// TIA Portal project "SzablonMASTER_V17" (V17)

(* hardware
DEVICE "S7-1200 station_1"  S7-1200 Station
   slot 0: "Rack_0"  Rack  V1.0
   slot 1: "PLC_1"  CPU 1214C DC/DC/DC  6ES7 214-1AG40-0XB0  V4.1
*)

// ===== PLC "PLC_1"  CPU 1214C DC/DC/DC =====

DATA_BLOCK "IO"   // DB1
{ S7_Optimized_Access := 'TRUE' }
VERSION : 0.1
   VAR
      StartS1 : Bool;
      StopS2 : Bool;
      RESETS3 : Bool;
      CzujnikEtykieciarkaB1 : Bool;
      CzujnikOdrzutB2 : Bool;
      CzujnikZbiornikB3 : Bool;
      CzujnikWieczkaB4 : Bool;
      SystemWizyjnyC1 : Bool;
      WagaC2 : Real;
      EtykieciarkaE1 : Bool;
      ZaworZ1 : Bool;
      SilownikA1 : Bool;
      SilownikA2 : Bool;
      PrzenosnikM1 : Bool;
      KolumnaZielonyH1 : Bool;
      KolumnaZoltyH2 : Bool;
      KolumnaCzerwonyH3 : Bool;
   END_VAR
BEGIN
END_DATA_BLOCK

DATA_BLOCK "ZadanieFinaloweMASTER_DB"   // DB2
{ S7_Optimized_Access := 'TRUE' }
VERSION : 0.1
// stored: InstanceOfName ZadanieFinaloweMASTER
"ZadanieFinaloweMASTER"
BEGIN
   StopS2 := true;
END_DATA_BLOCK

// folder: System blocks/Program resources

DATA_BLOCK "IEC_Timer_0_DB"   // DB3
{ S7_Optimized_Access := 'TRUE' }
AUTHOR : Simatic
FAMILY : IEC
NAME : IEC_TMR
VERSION : 1.0
// stored: InstanceOfName IEC_TIMER
"IEC_TIMER"
BEGIN
END_DATA_BLOCK

DATA_BLOCK "IEC_Timer_1_DB"   // DB4
{ S7_Optimized_Access := 'TRUE' }
AUTHOR : Simatic
FAMILY : IEC
NAME : IEC_TMR
VERSION : 1.0
// stored: InstanceOfName IEC_TIMER
"IEC_TIMER"
BEGIN
END_DATA_BLOCK

DATA_BLOCK "IEC_Timer_0_DB_1"   // DB5
{ S7_Optimized_Access := 'TRUE' }
AUTHOR : Simatic
FAMILY : IEC
NAME : IEC_TMR
VERSION : 1.0
// stored: InstanceOfName IEC_TIMER
"IEC_TIMER"
BEGIN
END_DATA_BLOCK

DATA_BLOCK "IEC_Timer_0_DB_2"   // DB6
{ S7_Optimized_Access := 'TRUE' }
AUTHOR : Simatic
FAMILY : IEC
NAME : IEC_TMR
VERSION : 1.0
// stored: InstanceOfName IEC_TIMER
"IEC_TIMER"
BEGIN
END_DATA_BLOCK

DATA_BLOCK "IEC_Counter_0_DB"   // DB7
{ S7_Optimized_Access := 'TRUE' }
AUTHOR : Simatic
FAMILY : IEC
NAME : CNTR
VERSION : 1.0
// stored: InstanceOfName IEC_COUNTER
"IEC_COUNTER"
BEGIN
END_DATA_BLOCK

DATA_BLOCK "IEC_Timer_0_DB_3"   // DB8
{ S7_Optimized_Access := 'TRUE' }
AUTHOR : Simatic
FAMILY : IEC
NAME : IEC_TMR
VERSION : 1.0
// stored: InstanceOfName IEC_TIMER
"IEC_TIMER"
BEGIN
END_DATA_BLOCK

// folder: (top level)

FUNCTION_BLOCK "ZadanieFinaloweMASTER"   // FB1, LAD
{ S7_Optimized_Access := 'TRUE' }
VERSION : 0.1
   VAR_INPUT
      StartS1 : Bool;
      StopS2 : Bool;
      RESETS3 : Bool;
      CzujnikEtykieciarkaB1 : Bool;
      CzujnikOdrzutB2 : Bool;
      CzujnikZbiornikB3 : Bool;
      CzujnikWieczkaB4 : Bool;
      SystemWizyjnyC1 : Bool;
      WagaC2 : Real;
   END_VAR
   VAR_OUTPUT
      EtykieciarkaE1 : Bool;
      ZaworZ1 : Bool;
      SilownikA1 : Bool;
      SilownikA2 : Bool;
      PrzenosnikM1 : Bool;
      KolumnaZielonyH1 : Bool;
      KolumnaZoltyH2 : Bool;
      KolumnaCzerwonyH3 : Bool;
   END_VAR
   VAR
      Run : Bool;
      Run_edgeP : Bool;
      Run_edgeN : Bool;
      T1_edge : Bool;
      A2_edge : Bool;
      B3_edge : Bool;
      B4_edge : Bool;
      WagaPuls : Bool;
      "WagaPuls edge" : Bool;
      Alarm : Bool;
      DB5_Q_edge : Bool;
   END_VAR
   VAR_TEMP
      T : Real;
      T_high : Real;
      T_Int : Int;
      T_high_Int : Int;
      Alarm_1_5Hz : Bool;
   END_VAR
   VAR_TEMP   // added for the SCL form of the ladder/FBD networks
      _w1 : Bool;
      _w2 : Bool;
   END_VAR
BEGIN

REGION Network 1
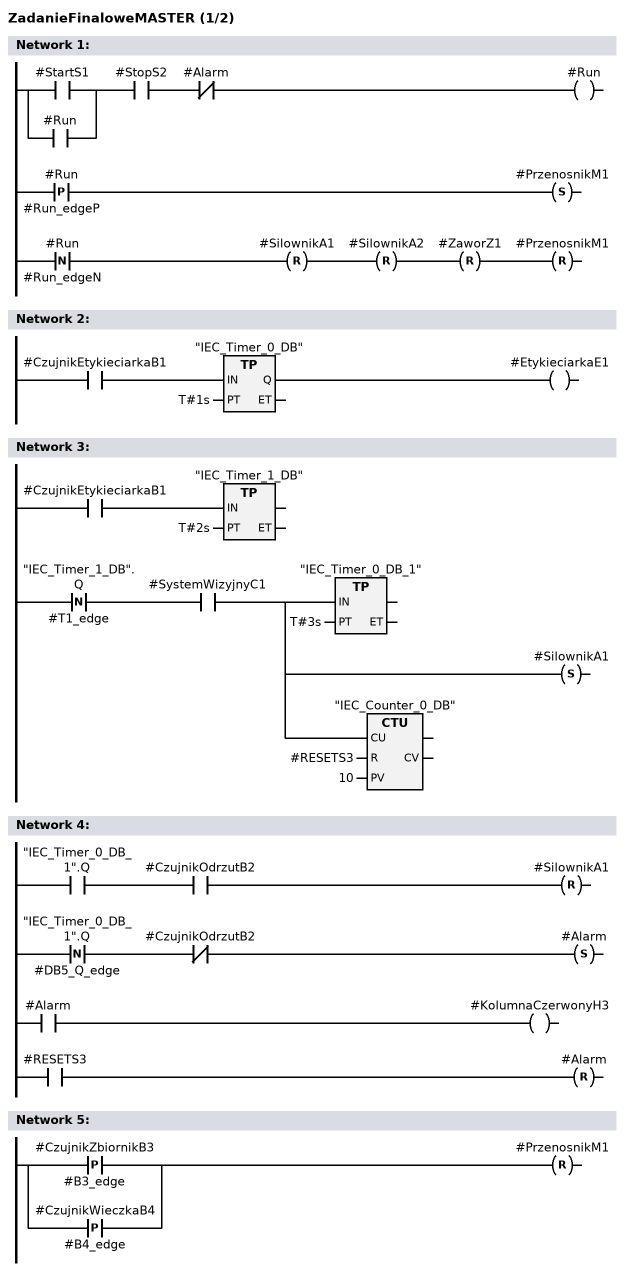
   RUNG wire#powerrail
      Contact( #StartS1 )
      wire#w1
      Contact( #StopS2 )
      I_Contact( #Alarm )
      Coil( #Run )
   END_RUNG
   RUNG wire#powerrail
      Contact( #Run )
   END_RUNG wire#w1
   RUNG wire#powerrail
      P_Contact(operand := #Run, bit := #Run_edgeP)
      S_Coil( #PrzenosnikM1 )
   END_RUNG
   RUNG wire#powerrail
      N_Contact(operand := #Run, bit := #Run_edgeN)
      R_Coil( #SilownikA1 )
      R_Coil( #SilownikA2 )
      R_Coil( #ZaworZ1 )
      R_Coil( #PrzenosnikM1 )
   END_RUNG
   // the same network as SCL:
   #Run := (#StartS1 OR #Run) AND #StopS2 AND NOT #Alarm;
   #_w1 := #Run AND NOT #Run_edgeP;   // rising edge of #Run
   #Run_edgeP := #Run;
   IF #_w1 THEN #PrzenosnikM1 := TRUE; END_IF;
   #_w2 := NOT #Run AND #Run_edgeN;   // falling edge of #Run
   #Run_edgeN := #Run;
   IF #_w2 THEN
       #SilownikA1 := FALSE;
       #SilownikA2 := FALSE;
       #ZaworZ1 := FALSE;
       #PrzenosnikM1 := FALSE;
   END_IF;
END_REGION

REGION Network 2
   "IEC_Timer_0_DB".TP(IN := #CzujnikEtykieciarkaB1, PT := T#1s);
   #EtykieciarkaE1 := "IEC_Timer_0_DB".Q;
END_REGION

REGION Network 3
   "IEC_Timer_1_DB".TP(IN := #CzujnikEtykieciarkaB1, PT := T#2s);
   #_w1 := NOT "IEC_Timer_1_DB".Q AND #T1_edge;   // falling edge of "IEC_Timer_1_DB".Q
   #T1_edge := "IEC_Timer_1_DB".Q;
   #_w2 := #_w1 AND #SystemWizyjnyC1;
   "IEC_Timer_0_DB_1".TP(IN := #_w2, PT := T#3s);
   IF #_w2 THEN #SilownikA1 := TRUE; END_IF;
   "IEC_Counter_0_DB".CTU(CU := #_w2, R := #RESETS3, PV := 10);
END_REGION

REGION Network 4
   RUNG wire#powerrail
      Contact( "IEC_Timer_0_DB_1".Q )
      Contact( #CzujnikOdrzutB2 )
      R_Coil( #SilownikA1 )
   END_RUNG
   RUNG wire#powerrail
      N_Contact(operand := "IEC_Timer_0_DB_1".Q, bit := #DB5_Q_edge)
      I_Contact( #CzujnikOdrzutB2 )
      S_Coil( #Alarm )
   END_RUNG
   RUNG wire#powerrail
      Contact( #Alarm )
      Coil( #KolumnaCzerwonyH3 )
   END_RUNG
   RUNG wire#powerrail
      Contact( #RESETS3 )
      R_Coil( #Alarm )
   END_RUNG
   // the same network as SCL:
   IF "IEC_Timer_0_DB_1".Q AND #CzujnikOdrzutB2 THEN #SilownikA1 := FALSE; END_IF;
   #_w1 := NOT "IEC_Timer_0_DB_1".Q AND #DB5_Q_edge;   // falling edge of "IEC_Timer_0_DB_1".Q
   #DB5_Q_edge := "IEC_Timer_0_DB_1".Q;
   IF #_w1 AND NOT #CzujnikOdrzutB2 THEN #Alarm := TRUE; END_IF;
   #KolumnaCzerwonyH3 := #Alarm;
   IF #RESETS3 THEN #Alarm := FALSE; END_IF;
END_REGION

REGION Network 5
   RUNG wire#powerrail
      P_Contact(operand := #CzujnikZbiornikB3, bit := #B3_edge)
      wire#w1
      R_Coil( #PrzenosnikM1 )
   END_RUNG
   RUNG wire#powerrail
      P_Contact(operand := #CzujnikWieczkaB4, bit := #B4_edge)
   END_RUNG wire#w1
   // the same network as SCL:
   #_w1 := #CzujnikZbiornikB3 AND NOT #B3_edge;   // rising edge of #CzujnikZbiornikB3
   #B3_edge := #CzujnikZbiornikB3;
   #_w2 := #CzujnikWieczkaB4 AND NOT #B4_edge;   // rising edge of #CzujnikWieczkaB4
   #B4_edge := #CzujnikWieczkaB4;
   IF #_w1 OR #_w2 THEN #PrzenosnikM1 := FALSE; END_IF;
END_REGION

REGION Network 6
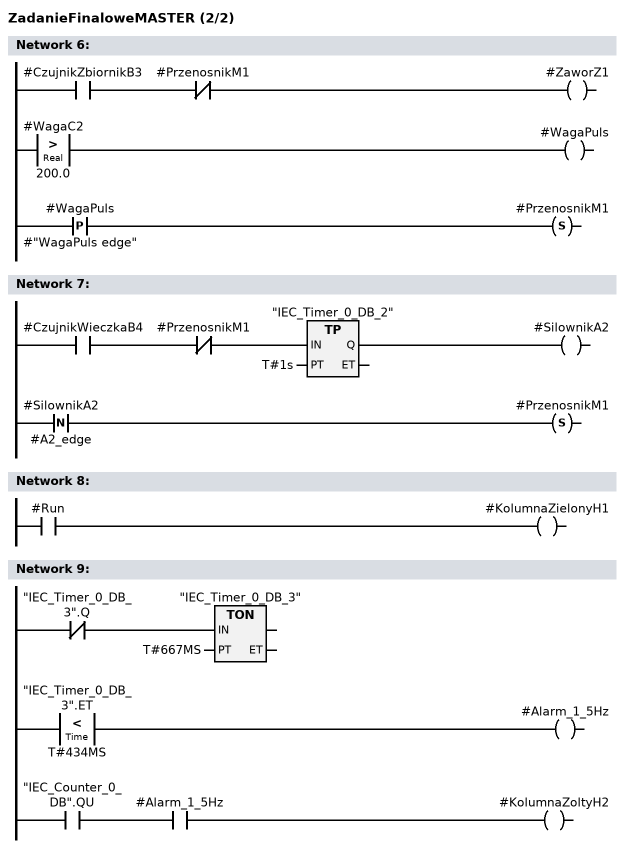
   RUNG wire#powerrail
      Contact( #CzujnikZbiornikB3 )
      I_Contact( #PrzenosnikM1 )
      Coil( #ZaworZ1 )
   END_RUNG
   RUNG wire#powerrail
      { S7_Templates := "SrcType := Real" } GT_Contact(in1 := #WagaC2, in2 := 200.0)
      Coil( #WagaPuls )
   END_RUNG
   RUNG wire#powerrail
      P_Contact(operand := #WagaPuls, bit := #"WagaPuls edge")
      S_Coil( #PrzenosnikM1 )
   END_RUNG
   // the same network as SCL:
   #ZaworZ1 := #CzujnikZbiornikB3 AND NOT #PrzenosnikM1;
   #WagaPuls := #WagaC2 > 200.0;
   #_w1 := #WagaPuls AND NOT #"WagaPuls edge";   // rising edge of #WagaPuls
   #"WagaPuls edge" := #WagaPuls;
   IF #_w1 THEN #PrzenosnikM1 := TRUE; END_IF;
END_REGION

REGION Network 7
   "IEC_Timer_0_DB_2".TP(IN := #CzujnikWieczkaB4 AND NOT #PrzenosnikM1, PT := T#1s);
   #SilownikA2 := "IEC_Timer_0_DB_2".Q;
   #_w1 := NOT #SilownikA2 AND #A2_edge;   // falling edge of #SilownikA2
   #A2_edge := #SilownikA2;
   IF #_w1 THEN #PrzenosnikM1 := TRUE; END_IF;
END_REGION

REGION Network 8
   RUNG wire#powerrail
      Contact( #Run )
      Coil( #KolumnaZielonyH1 )
   END_RUNG
   // the same network as SCL:
   #KolumnaZielonyH1 := #Run;
END_REGION

REGION Network 9
   "IEC_Timer_0_DB_3".TON(IN := NOT "IEC_Timer_0_DB_3".Q, PT := T#667MS);
   #Alarm_1_5Hz := "IEC_Timer_0_DB_3".ET < T#434MS;
   #KolumnaZoltyH2 := "IEC_Counter_0_DB".QU AND #Alarm_1_5Hz;
END_REGION
END_FUNCTION_BLOCK

ORGANIZATION_BLOCK "Main"   // OB1, LAD, ProgramCycle
TITLE = "Main Program Sweep (Cycle)"
{ S7_Optimized_Access := 'TRUE' }
VERSION : 0.1
   VAR_INPUT
      Initial_Call : Bool;   // Initial call of this OB
      Remanence : Bool;   // =True, if remanent data are available
   END_VAR
BEGIN

REGION Network 1: Zadanie finałowe kategorii MASTER
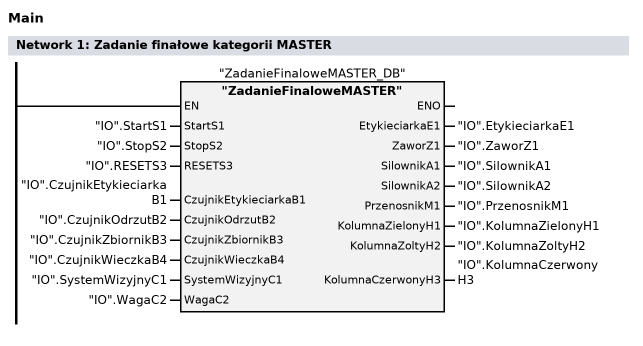
   RUNG wire#powerrail
      "ZadanieFinaloweMASTER_DB"(StartS1 := "IO".StartS1, StopS2 := "IO".StopS2, RESETS3 := "IO".RESETS3, CzujnikEtykieciarkaB1 := "IO".CzujnikEtykieciarkaB1, CzujnikOdrzutB2 := "IO".CzujnikOdrzutB2, CzujnikZbiornikB3 := "IO".CzujnikZbiornikB3, CzujnikWieczkaB4 := "IO".CzujnikWieczkaB4, SystemWizyjnyC1 := "IO".SystemWizyjnyC1, WagaC2 := "IO".WagaC2, EtykieciarkaE1 => "IO".EtykieciarkaE1, ZaworZ1 => "IO".ZaworZ1, SilownikA1 => "IO".SilownikA1, SilownikA2 => "IO".SilownikA2, PrzenosnikM1 => "IO".PrzenosnikM1, KolumnaZielonyH1 => "IO".KolumnaZielonyH1, KolumnaZoltyH2 => "IO".KolumnaZoltyH2, KolumnaCzerwonyH3 => "IO".KolumnaCzerwonyH3)
   END_RUNG
   // the same network as SCL:
   "ZadanieFinaloweMASTER_DB"(StartS1 := "IO".StartS1,   // "ZadanieFinaloweMASTER"
                           StopS2 := "IO".StopS2,
                           RESETS3 := "IO".RESETS3,
                           CzujnikEtykieciarkaB1 := "IO".CzujnikEtykieciarkaB1,
                           CzujnikOdrzutB2 := "IO".CzujnikOdrzutB2,
                           CzujnikZbiornikB3 := "IO".CzujnikZbiornikB3,
                           CzujnikWieczkaB4 := "IO".CzujnikWieczkaB4,
                           SystemWizyjnyC1 := "IO".SystemWizyjnyC1,
                           WagaC2 := "IO".WagaC2,
                           EtykieciarkaE1 => "IO".EtykieciarkaE1,
                           ZaworZ1 => "IO".ZaworZ1,
                           SilownikA1 => "IO".SilownikA1,
                           SilownikA2 => "IO".SilownikA2,
                           PrzenosnikM1 => "IO".PrzenosnikM1,
                           KolumnaZielonyH1 => "IO".KolumnaZielonyH1,
                           KolumnaZoltyH2 => "IO".KolumnaZoltyH2,
                           KolumnaCzerwonyH3 => "IO".KolumnaCzerwonyH3);
END_REGION
END_ORGANIZATION_BLOCK